TYPE Vector3Position_typ :
STRUCT
	X		: LREAL;
	Y		: LREAL;
	Z		: LREAL;
END_STRUCT
END_TYPE

(* stored: Version 1.1.0.1, ProductVersion 3.1.4024.11
   DUT Vector3Position_typ: Id {59e1fcf7-162b-42cb-874e-d9abf930f135} *)
